(*			
	EVERDE sp. z o.o.
	Rafał Osajda		16.07.2025		TC 4024.66
	Lampka rozszerzona o moduł FB_Impuls co integruje w niej możlwiość mgania lub świecenie ciągłego
*)
FUNCTION_BLOCK FB_LampkaRozszerzona EXTENDS FB_Lampka IMPLEMENTS ITF_LampkaRozszerzona
VAR
	fbImpuls				: B_Baza.FB_Impuls;
END_VAR

METHOD PUBLIC Ciagly
VAR_INPUT
	bIN				: BOOL;
END_VAR
THIS^.fbImpuls.Ciagly (bIN			:= bIN);
END_METHOD

(*			
	EVERDE sp. z o.o.
	Rafał Osajda		31.01.2025		TC 4026.13		wer. 0.0.0.1
	Sterowanie działem ipulsatora 
*)
METHOD PUBLIC Migaj
VAR_INPUT
	bIN				: bool;
END_VAR
THIS^.fbImpuls.Migaj (bIN	:= bIN);
END_METHOD

METHOD PUBLIC Reset
VAR_INPUT
END_VAR
THIS^.fbImpuls.Reset ();
END_METHOD

(*			
	EVERDE sp. z o.o.
	Rafał Osajda		05.02.2025		TC 4026.13		wer. 0.0.0.1
	Zwraca czy lampka wlaczona
*)
METHOD Stan : BOOL
Stan					:= SUPER^.Stan ();
END_METHOD

(*			
	EVERDE sp. z o.o.
	Rafał Osajda		05.02.2025		TC 4026.13		wer. 0.0.0.1
	Sterowanie swieceniem lampki - włącz/wyłącz
*)
METHOD Steruj
VAR_INPUT
	bIN	: BOOL;
END_VAR
IF (bIN) THEN
	THIS^.fbImpuls.Wlacz (bSwiec := TRUE, bMigaj := TRUE, tWlaczony := T#0S, tWylaczony := T#0S);
ELSE
	THIS^.fbImpuls.Wylacz ();
END_IF
END_METHOD

(*			
	EVERDE sp. z o.o.
	Rafał Osajda		31.01.2025		TC 4026.13		wer. 0.0.0.1
	
*)
METHOD PUBLIC ustawCzasZapalony
VAR_INPUT
	tIN						: TIME;
END_VAR
THIS^.fbImpuls.ustawCzasZapalony (tIN				:= tIN);
END_METHOD

(*			
	EVERDE sp. z o.o.
	Rafał Osajda		31.01.2025		TC 4026.13		wer. 0.0.0.1
	Ustawia czas zgaszonej lampki
*)
METHOD PUBLIC ustawCzasZgaszony
VAR_INPUT
	tIN					: TIME;
END_VAR
THIS^.fbImpuls.ustawCzasZgaszony (tIN			:= tIN);
END_METHOD

(*			
	EVERDE sp. z o.o.
	Rafał Osajda		05.02.2025		TC 4026.13		wer. 0.0.0.1
	Wlacza lampke - praca ciągła
*)
METHOD Wlacz
THIS^.fbImpuls.Wlacz (bSwiec := TRUE, bMigaj := TRUE, tWlaczony := T#0S, tWylaczony := T#0S);
END_METHOD

METHOD PUBLIC Wlacz2
VAR_INPUT
	bSwiec		: BOOL;
	bMigaj		: BOOL;
	tWlaczony	: TIME;
	tWylaczony	: TIME;
END_VAR
THIS^.fbImpuls.Wlacz (
	bSwiec		:= bSwiec,
	bMigaj		:= bMigaj,
	tWlaczony	:= tWlaczony,
	tWylaczony	:= tWylaczony
);
END_METHOD

(*			
	EVERDE sp. z o.o.
	Rafał Osajda		27.03.2025		TC 4024.66
	Wywolanie co cykl operacji 
*)
METHOD PUBLIC WykonywaneCoCykl_Operacje
VAR_INPUT
END_VAR
SUPER^.WykonywaneCoCykl_Operacje ();

THIS^.fbImpuls ();
END_METHOD

(*			
	EVERDE sp. z o.o.
	Rafał Osajda		27.03.2025		TC 4024.66
	Aktualizacja flag 
*)
METHOD PUBLIC WykonywaneCoCykl_Status
VAR_INST
END_VAR
SUPER^.WykonywaneCoCykl_Status ();

//SUPER^.Steruj (bIN := THIS^.fbImpuls.Stan ());
THIS^.bLampka		:= THIS^.fbImpuls.Stan ();
END_METHOD

(*			
	EVERDE sp. z o.o.
	Rafał Osajda		05.02.2025		TC 4026.13		wer. 0.0.0.1
	Wylacza lampke
*)
METHOD Wylacz
THIS^.fbImpuls.Wylacz ();
END_METHOD

END_FUNCTION_BLOCK

(* stored: Version 1.1.0.1
   POU FB_LampkaRozszerzona: Id {dcff81a1-6dd7-4eaf-907a-2248d98a1fd0}, SpecialFunc None
   Folder Impuls: Id {00302c85-f7fe-4010-b913-cb28ac209e80}
   Folder Lampka: Id {1ce39044-512f-4976-97b5-7f5d1cfcc4ca}
   Method Ciagly: Id {d73aa7c8-66fb-44b9-abcb-6defbf850207}
   Method Migaj: Id {7308fc6d-0df1-0fc9-3448-90bfe4f60c6d}
   Method Reset: Id {6adcf835-6ae6-41e9-928f-14ae42082f84}
   Method Stan: Id {ee9e61ef-6944-415e-a33e-67301498eb26}
   Method Steruj: Id {f185e64f-f3ee-4960-826a-7adb0ab287d7}
   Method ustawCzasZapalony: Id {6984913b-06ff-0018-00ab-a77455e9d2b1}
   Method ustawCzasZgaszony: Id {6e8b987e-d352-044d-0d8b-d018d73edb47}
   Method Wlacz: Id {3cba340c-0e1a-4db9-b5dc-78c607c4f1e1}
   Method Wlacz2: Id {394fd72e-1ef7-4d61-b407-9f1d7f9d1d0d}
   Method WykonywaneCoCykl_Operacje: Id {3122b5f5-fb1e-4355-b29b-0ca3046f4573}
   Method WykonywaneCoCykl_Status: Id {22023be3-3f2d-479c-beea-467a1af9fb42}
   Method Wylacz: Id {74da1db2-cae1-4989-b15d-2e841810dcc3} *)
